Fanuc KAREL source: GET_TSK_INFO.kl

PROGRAM T
%NOLOCKGROUP
VAR
 v0 : STRING[40]
 v1 : INTEGER
 v2 : INTEGER
 v3 : INTEGER
 v4 : STRING[40]
 v5 : INTEGER
BEGIN
 GET_TSK_INFO(v0, v1, v2, v3, v4, v5)
END T
